// TIA Portal V16 export
// export: Created 2023-05-08T20:46:19.4733709Z, ExportSetting WithDefaults, DisplayName Totally Integrated Automation Portal, DisplayVersion V16 Update 6, DisplayName TIA Portal Version Control Interface, DisplayVersion V16 Update 2, DisplayName TIA Portal Openness, DisplayVersion V16 Update 6, DisplayName STEP 7 Professional, DisplayVersion V16 Update 6, DisplayName STEP 7 Safety, DisplayVersion V16, DisplayName WinCC Advanced, DisplayVersion V16 Update 6
ORGANIZATION_BLOCK "Main"   // OB1, SCL, ProgramCycle
TITLE = "Main Program Sweep (Cycle)"
{ S7_Optimized_Access := 'TRUE' }
VERSION : 0.1
// stored: AutoNumber true, IsIECCheckEnabled false, SetENOAutomatically false
   VAR_INPUT
      Initial_Call : Bool;   // Initial call of this OB
      Remanence : Bool;   // =True, if remanent data are available
   END_VAR
BEGIN

   "MHJ-PLC-Lab-Function-S71500"(MinDiByte:=0,
                                 MaxDiByte:=1);
   "MHJ-PLC-Lab-Function-S71500-NextInputArea"(MinDiByte:=256,
                                               MaxDiByte:=259);


   "K1" := "S2";
   "K2" := "S3";
   "P5" := "S1";
   "P4" := "S4";
   "P3" := "S3";
   "P2" := NOT "S0";
   "P1" := "S3";
   "IstPos" := "SollPos";
END_ORGANIZATION_BLOCK
